FUNCTION_BLOCK COURIER_CAT_HMI (* Service Interface Function Block Type *)
  (* Standard: 61499-2 *)
  (* Version 0.0, 12/17/2022, Dmitrii, Flexbridge AB, template *)
  PACKAGE Main;
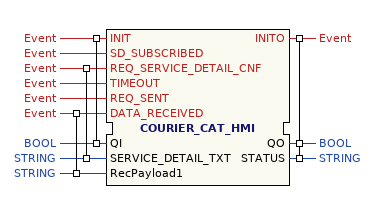
  EVENT_INPUT
    INIT WITH QI;
    SD_SUBSCRIBED;
    REQ_SERVICE_DETAIL_CNF WITH SERVICE_DETAIL_TXT;
    TIMEOUT;
    REQ_SENT;
    DATA_RECEIVED WITH RecPayload1;
  END_EVENT
  EVENT_OUTPUT
    INITO WITH QO, STATUS;
  END_EVENT
  VAR_INPUT
    QI : BOOL;
    SERVICE_DETAIL_TXT : STRING;
    RecPayload1 : STRING;
  END_VAR
  VAR_OUTPUT
    QO : BOOL; (* Event Output Qualifier *)
    STATUS : STRING; (* Service Status *)
  END_VAR
  SERVICE /
    SEQUENCE 
    END_SEQUENCE
  END_SERVICE
END_FUNCTION_BLOCK
